// TIA Portal V18 export
DATA_BLOCK "Block_1_DB_2"   // DB36
// stored: InstanceOfName Block_1, InstanceOfType FB
"Block_1"
   // VAR_INPUT
   //    Input_1 : Bool;
   // END_VAR
   // VAR
   //    Test_Mode : Word;
   //    "Counter" : Word;
   //    Delay_Timer { S7_SetPoint := 'True'} : TON_TIME;
   //    TurnOnOffTimer { S7_SetPoint := 'True'} : Bool;
   // END_VAR
BEGIN
END_DATA_BLOCK
